FUNCTION_BLOCK TcoTixonPickVibroBasic_v_1_x_x EXTENDS TcoCore.TcoComponent
VAR_INPUT
    inControllerInAuto : BOOL;
    inNotEmptyFeeder : BOOL;
    inSeparatorHomePos : BOOL;
    inFillingSensor : BOOL;
    inSeparatorPresent : BOOL;
    inSeparatorWorkPos : BOOL;
    inPickZone : BOOL;
END_VAR
VAR_OUTPUT
    outFeedingA : BOOL;
    outSepareComponent : BOOL;
    outBlowValveA : BOOL;
    outRedLed : BOOL;
    outGreenLed : BOOL;
    outHopper : BOOL;
END_VAR
VAR
    {attribute addProperty Name "<#Status#>"}
    {attribute clr [ReadOnly()]}
    _status : TcoTixonPickVibroBasic_Status_v_1_x_x;
    {attribute addProperty Name "<#Control#>"}
    _control : TcoTixonPickVibroBasic_Control_v_1_x_x;
    {attribute addProperty Name "<#Config#>"}
    _config : TcoTixonPickVibroBasic_Config_v_1_x_x;
    _someTaskIsActive : BOOL;
    {attribute 'hide'}
    _blink : TcoUtilities.TcoBlinker(THIS^);
    _runAutomatic : BOOL;
    _hasError : BOOL;
END_VAR
VAR
    {attribute addProperty Name "<#Separator task#>"}
    _separatorTask : TcoTixonPickVibroBasicSeparatorTask(THIS^);
    {attribute addProperty Name "<#Buffer task#>"}
    _bufferTask : TcoTixonBufferTask(THIS^);
    {attribute addProperty Name "<#Hopper task#>"}
    _hopperTask : TcoTixonHopperTask(THIS^);
    {attribute addProperty Name "<#Restore#>"}
    _restoreTask : TcoCore.TcoTask(THIS^);
END_VAR
VAR
    {attribute 'hide'}
    _sb : TcoCore.StringBuilder;
END_VAR

_blink(inOnTime := _config.BlinkTime, inOffTime := _config.BlinkTime);
UpdateStatus();
_separatorTask.Enabled := TRUE;
_separatorTask(inoConfig := _config, inoControl := _control, inoStatus := _status);
_bufferTask.Enabled := TRUE;
_bufferTask(inoConfig := _config, inoControl := _control, inoStatus := _status);
_hopperTask.Enabled := _config.HopperActive;
_hopperTask(inoConfig := _config, inoControl := _control, inoStatus := _status);
//*************RESTORE********************
_restoreTask.Enabled := TRUE;

IF _restoreTask.Execute() THEN
    Restore();
    _restoreTask.DoneWhen(TRUE);
END_IF
//****************************************
UpdateControl();

METHOD PUBLIC BufferFeed : TcoCore.ITcoTaskStatus
BufferFeed := _bufferTask.Invoke();
_bufferTask.AutoRestore := false;
END_METHOD

PROPERTY PUBLIC BufferTask : REFERENCE TO TcoTixonBufferTask
GET
BufferTask ref= _bufferTask;
END_GET
END_PROPERTY

(*~
    <docu>
        <summary>
            Gets the configuration of the Tixon Step.
        </summary>
    </docu>
~*)
PROPERTY Config : REFERENCE TO TcoTixonPickVibroBasic_Config_v_1_x_x
GET
Config REF= _config;
END_GET
END_PROPERTY

METHOD PUBLIC CyclicBufferFeed : TcoCore.ITcoTaskStatus
CyclicBufferFeed := _bufferTask.Invoke();
_bufferTask.AutoRestore := true;
END_METHOD

METHOD PUBLIC CyclicHopperFeed : TcoCore.ITcoTaskStatus
CyclicHopperFeed := _hopperTask.Invoke();
_hopperTask.AutoRestore := TRUE;
END_METHOD

METHOD PUBLIC CyclicSepare : TcoCore.ITcoTaskStatus
CyclicSepare := _separatorTask.Invoke();
_separatorTask.AutoRestore := true;
END_METHOD

METHOD PUBLIC DefaultSignalisation
VAR_INPUT
END_VAR
// led signalisation
_hasError := _separatorTask.Error OR _bufferTask.Error OR _hopperTask.Error;
_control.GreenLed := FALSE;
_control.RedLed := FALSE;

IF NOT _status.ControllerInAuto THEN
    _control.GreenLed := TRUE;
    _control.RedLed := TRUE;
ELSIF _hasError AND _blink.IsOn AND _status.ControllerInAuto THEN
    _control.RedLed := TRUE;
ELSIF _status.ControllerInAuto AND NOT _hasError AND _status.NotEmptyFeeder THEN
    _control.GreenLed := TRUE;
ELSIF _blink.IsOn AND _status.ControllerInAuto AND NOT _status.NotEmptyFeeder THEN
    _control.GreenLed := TRUE;
    _control.RedLed := TRUE;
END_IF
END_METHOD

METHOD PUBLIC HopperFeed : TcoCore.ITcoTaskStatus
HopperFeed := _hopperTask.Invoke();
_hopperTask.AutoRestore := false;
END_METHOD

PROPERTY PUBLIC HopperTask : reference TO TcoTixonHopperTask
GET
HopperTask ref= _hopperTask;
END_GET
END_PROPERTY

(*~
    <docu>
        <summary>
            Restores this instance to the Ready state. Can be called explicitly or from within one of the restore mechanisms.
        </summary>
    </docu>
~*)
METHOD Restore : ITcoRestorable
RestoreTasks();
_control.BlowAValve := FALSE;
_control.FeedingA := FALSE;
_control.GreenLed := FALSE;
_control.RedLed := FALSE;
_control.SepareComponent := FALSE;
_control.Hooper := FALSE;
END_METHOD

METHOD INTERNAL RestoreTasks
//_resetTask.Restore();
_separatorTask.Restore();
_bufferTask.Restore();
_hopperTask.Restore();
END_METHOD

PROPERTY PUBLIC SeparatorTask : REFERENCE TO TcoTixonPickVibroBasicSeparatorTask
GET
SeparatorTask ref= _separatorTask;
END_GET
END_PROPERTY

METHOD PUBLIC Separe : TcoCore.ITcoTaskStatus
Separe := _separatorTask.Invoke();
_separatorTask.AutoRestore := false;
END_METHOD

(*~
    <docu>
        <summary>
            Custom service (manual, maintenance) logic.
            This method must be implemented in derived class.
        </summary>
    </docu>
~*)
METHOD PROTECTED ServiceMode
END_METHOD

(*~
    <docu>
        <summary>
            Gets the status of the Tixon Step.
        </summary>
    </docu>
~*)
PROPERTY Status : REFERENCE TO TcoTixonPickVibroBasic_Status_v_1_x_x
GET
Status REF= _status;
END_GET
END_PROPERTY

METHOD INTERNAL UpdateControl
VAR_INPUT
END_VAR
VAR
    index : INT;
END_VAR
outBlowValveA := _control.BlowAValve;
outFeedingA := _control.FeedingA;
outGreenLed := _control.GreenLed;
outRedLed := _control.RedLed;
outSepareComponent := _control.SepareComponent;
outHopper := _control.Hooper;
END_METHOD

METHOD INTERNAL UpdateStatus
VAR
END_VAR
_status.NotEmptyFeeder := inNotEmptyFeeder;
_status.SeparatorHomePos := inSeparatorHomePos;
_status.SeparatorPresent := inSeparatorPresent;
_status.FillingSensor := inFillingSensor;
_status.SeparatorWorkPos := inSeparatorWorkPos;
_status.ControllerInAuto := inControllerInAuto;
_status.InPickZone := inPickZone;
END_METHOD

END_FUNCTION_BLOCK

(* stored: Version 1.1.0.1, ProductVersion 3.1.4024.12
   POU TcoTixonPickVibroBasic_v_1_x_x: Id {83547b0c-58d3-06f9-24e8-4f9babe79f42}, SpecialFunc None
   Folder Operations: Id {6ce7b4b4-b012-0f38-137e-787f453be3fb}
   Folder Loop: Id {6bb60c61-d3b8-0669-3372-883cf243e584}
   Folder Single: Id {3973f039-9330-02d6-1985-259c1f5c6b50}
   Folder Task: Id {e73ae2b2-cc40-061e-090b-0c49a25786e8}
   Method BufferFeed: Id {50330b28-f6db-0c43-38a7-31a9c7311142}
   Property BufferTask: Id {4d9c6cd9-ae31-0481-2daf-b20453218bd2}
   Get Get: Id {7a506f2a-9a2e-0542-3144-a4171c920bc1}
   Property Config: Id {88c4ce96-49c2-071e-0a2b-c2d5e392553b}
   Get Get: Id {37ea61ff-f0c1-01c9-32e2-89ab657135f9}
   Method CyclicBufferFeed: Id {d5016904-a61c-0cba-1fa9-efab402f6568}
   Method CyclicHopperFeed: Id {1c7c347c-d89d-0801-0a82-6aac33a5008a}
   Method CyclicSepare: Id {e9888e68-476c-0a72-3a60-609cf2730ac3}
   Method DefaultSignalisation: Id {4e87b105-2825-0988-259f-958cf61d9220}
   Method HopperFeed: Id {73811985-0061-0629-034b-5f32c108c269}
   Property HopperTask: Id {0245b470-b2fa-0e82-20fc-bb3fd02abb0d}
   Get Get: Id {728a3245-547e-095b-18f2-d42a3022f167}
   Method Restore: Id {3b219525-b670-00c2-3709-74790d8af120}
   Method RestoreTasks: Id {cdb3c77d-1f2c-0a5a-0aaf-fbebc77a73a6}
   Property SeparatorTask: Id {2bed9c28-fe4b-05ed-2432-bb1aed87a6c6}
   Get Get: Id {9c9f9bb7-ce1e-04ff-09a6-f8240ed6fdb1}
   Method Separe: Id {0a21eba1-5f9b-081f-0db4-b4b909bbbebc}
   Method ServiceMode: Id {11df6814-169b-0a60-108c-99fd7081fd04}
   Property Status: Id {742b1bf2-4e6b-0670-188b-2e9c44331153}
   Get Get: Id {cc51ddc1-9c84-0e2b-1ca2-d826dae1777a}
   Method UpdateControl: Id {c0b8ec0c-e63a-09bd-0a8a-33a90cf28e30}
   Method UpdateStatus: Id {d2a4a8ea-78a1-093a-2453-b7243b379bec} *)
